{attribute 'qualified_only'}
VAR_GLOBAL
END_VAR

(* stored: Version 1.1.0.1, ProductVersion 3.1.4024.16
   GVL branch: Id {1ff9164b-c251-42d9-a934-311393f44799} *)
